(* CoDeSys 2.3 export: F_WRITE_SENSOR_KG.EXP *)

(* POU FUN/PARAMETERS/F_WRITE_SENSOR_KG, ST *)
FUNCTION F_WRITE_SENSOR_KG : BOOL
VAR_INPUT
	wSize   :DWORD;
	pBuffer :POINTER TO BYTE;
END_VAR
VAR_IN_OUT
	wPos     : DWORD;
	stSensor : ST_SENSOR_KG;
END_VAR
VAR
END_VAR
F_ADD_STRINGX4_TO_BUFFER( S1:= CONCAT(stSensor.Name, '_K' ), S2:='$t', S3:= REAL_TO_STRING( stSensor.Cal_K ), S4:='$n', wSize := wSize, pBuffer := pBuffer, wPos := wPos );
F_ADD_STRINGX4_TO_BUFFER( S1:= CONCAT(stSensor.Name, '_C' ), S2:='$t', S3:= REAL_TO_STRING( stSensor.Cal_C ), S4:='$n', wSize := wSize, pBuffer := pBuffer, wPos := wPos );
END_FUNCTION
